(* PLC project  *)

PROGRAM P
  VAR  (* added by the conversion: wires and edge detectors of the diagram *)
    _F_SPLIT3_R : ANY;
    _F_SPLIT3_OUT : ANY;
  END_VAR

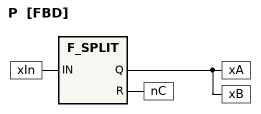
(* FBD diagram, written out as Structured Text *)
_F_SPLIT3_OUT := F_SPLIT(IN := xIn, R => _F_SPLIT3_R);
xA := _F_SPLIT3_OUT;
xB := _F_SPLIT3_OUT;
nC := _F_SPLIT3_R;
END_PROGRAM
